Staubli VAL3: onF6Event.pgx

program onF6Event(bool& l_bSave[])
  local bool l_bYes
  local string l_sMessage
  local string l_sButton[2]
  local num l_nResult
begin
  // look if the bButton is enable
  if bButton[5]
    //
    // Delete the select Item
    //
    call language:message(l_sMessage,80)
    // get the yes_no button Key
    call language:getYesNo(l_sButton)
    // ask the question
    call use:yes_no(l_sMessage,l_sButton,l_bYes)
    if l_bYes
      call prog:deleteItem(nIndex,l_nResult)
      // go back by one
      if nIndex>0
        nSelected=nId-1
      endIf
      call buildList()
      l_bSave=true
    endIf
  endIf
end
